INTERFACE I_HandoverEmulationListener

METHOD M_HandoverStartEvent
END_METHOD

END_INTERFACE

(* stored: Version 1.1.0.1, ProductVersion 3.1.4022.12
   Itf I_HandoverEmulationListener: Id {3c9120bb-8369-45ac-b8fa-2f0f357dfd44}
   Method M_HandoverStartEvent: Id {d0b4c508-af0a-478b-bfaa-a163cdeda0c0} *)
